FUNCTION_BLOCK Velocity_PI_LREAL3 (* Composite Function Block Type *)
  (* Standard: 61499-2 *)
  (* Version 0.0, 2018-07-28, 4DIAC-IDE, 4DIAC-Consortium *)
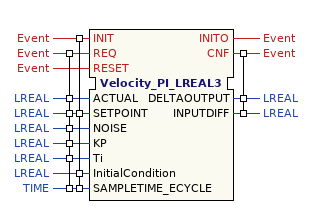
  EVENT_INPUT
    INIT WITH SAMPLETIME_ECYCLE, SETPOINT, InitialCondition; (* Initialization Request *)
    REQ WITH SAMPLETIME_ECYCLE, ACTUAL, SETPOINT, NOISE, KP, Ti; (* Normal Execution Request. disambung Event Cycle juga ya *)
    RESET;
  END_EVENT
  EVENT_OUTPUT
    INITO; (* Initialization Confirm *)
    CNF WITH DELTAOUTPUT, INPUTDIFF; (* Execution Confirmation *)
  END_EVENT
  VAR_INPUT
    ACTUAL : LREAL;
    SETPOINT : LREAL;
    NOISE : LREAL;
    KP : LREAL;
    Ti : LREAL;
    InitialCondition : LREAL;
    SAMPLETIME_ECYCLE : TIME;
  END_VAR
  VAR_OUTPUT
    DELTAOUTPUT : LREAL;
    INPUTDIFF : LREAL;
  END_VAR
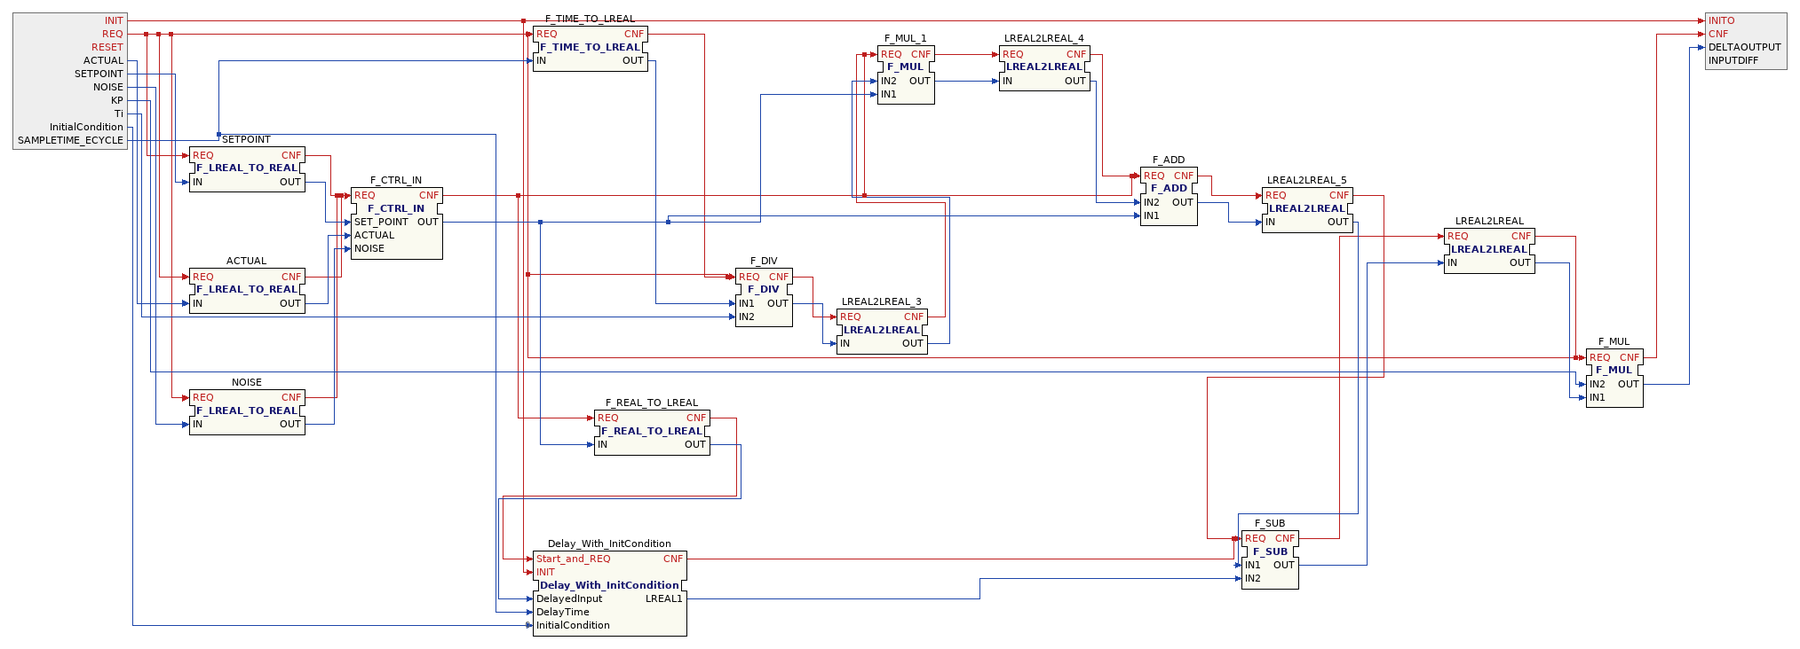
  FBS
    F_CTRL_IN : F_CTRL_IN;
    F_SUB : F_SUB;
    F_MUL : F_MUL;
    F_ADD : F_ADD;
    F_MUL_1 : F_MUL;
    F_DIV : F_DIV;
    SETPOINT : F_LREAL_TO_REAL;
    ACTUAL : F_LREAL_TO_REAL;
    NOISE : F_LREAL_TO_REAL;
    F_TIME_TO_LREAL : F_TIME_TO_LREAL;
    Delay_With_InitCondition : Delay_With_InitCondition(InitialCondition := 0);
    F_REAL_TO_LREAL : F_REAL_TO_LREAL;
    LREAL2LREAL_3 : LREAL2LREAL;
    LREAL2LREAL_5 : LREAL2LREAL;
    LREAL2LREAL_4 : LREAL2LREAL;
    LREAL2LREAL : LREAL2LREAL;
  END_FBS
  EVENT_CONNECTIONS
    F_MUL.CNF TO CNF;
    REQ TO SETPOINT.REQ;
    SETPOINT.CNF TO F_CTRL_IN.REQ;
    REQ TO ACTUAL.REQ;
    ACTUAL.CNF TO F_CTRL_IN.REQ;
    REQ TO NOISE.REQ;
    NOISE.CNF TO F_CTRL_IN.REQ;
    F_TIME_TO_LREAL.CNF TO F_DIV.REQ;
    REQ TO F_TIME_TO_LREAL.REQ;
    F_REAL_TO_LREAL.CNF TO Delay_With_InitCondition.Start_and_REQ;
    F_CTRL_IN.CNF TO F_REAL_TO_LREAL.REQ;
    INIT TO Delay_With_InitCondition.INIT;
    INIT TO INITO;
    LREAL2LREAL_3.CNF TO F_MUL_1.REQ;
    F_DIV.CNF TO LREAL2LREAL_3.REQ;
    F_ADD.CNF TO LREAL2LREAL_5.REQ;
    LREAL2LREAL_5.CNF TO F_SUB.REQ;
    REQ TO F_DIV.REQ;
    REQ TO F_MUL.REQ;
    Delay_With_InitCondition.CNF TO F_SUB.REQ;
    F_MUL_1.CNF TO LREAL2LREAL_4.REQ;
    LREAL2LREAL_4.CNF TO F_ADD.REQ;
    F_CTRL_IN.CNF TO F_ADD.REQ;
    F_CTRL_IN.CNF TO F_MUL_1.REQ;
    LREAL2LREAL.CNF TO F_MUL.REQ;
    F_SUB.CNF TO LREAL2LREAL.REQ;
  END_CONNECTIONS
  DATA_CONNECTIONS
    SETPOINT.OUT TO F_CTRL_IN.SET_POINT;
    SETPOINT TO SETPOINT.IN;
    ACTUAL TO ACTUAL.IN;
    ACTUAL.OUT TO F_CTRL_IN.ACTUAL;
    NOISE.OUT TO F_CTRL_IN.NOISE;
    NOISE TO NOISE.IN;
    SAMPLETIME_ECYCLE TO F_TIME_TO_LREAL.IN;
    F_TIME_TO_LREAL.OUT TO F_DIV.IN1;
    F_REAL_TO_LREAL.OUT TO Delay_With_InitCondition.DelayedInput;
    F_CTRL_IN.OUT TO F_REAL_TO_LREAL.IN;
    SAMPLETIME_ECYCLE TO Delay_With_InitCondition.DelayTime;
    F_DIV.OUT TO LREAL2LREAL_3.IN;
    LREAL2LREAL_3.OUT TO F_MUL_1.IN2;
    LREAL2LREAL_5.OUT TO F_SUB.IN1;
    F_ADD.OUT TO LREAL2LREAL_5.IN;
    F_MUL.OUT TO DELTAOUTPUT;
    InitialCondition TO Delay_With_InitCondition.InitialCondition;
    Ti TO F_DIV.IN2;
    KP TO F_MUL.IN2;
    Delay_With_InitCondition.LREAL1 TO F_SUB.IN2;
    F_MUL_1.OUT TO LREAL2LREAL_4.IN;
    LREAL2LREAL_4.OUT TO F_ADD.IN2;
    F_CTRL_IN.OUT TO F_ADD.IN1;
    F_CTRL_IN.OUT TO F_MUL_1.IN1;
    F_SUB.OUT TO LREAL2LREAL.IN;
    LREAL2LREAL.OUT TO F_MUL.IN1;
  END_CONNECTIONS
END_FUNCTION_BLOCK
